TYPE Recipe :
STRUCT
	aRecipe		: ARRAY[1..GVL_CONSTANT.MaxRecipeStep] OF RecipeStep; //Recipe Structure
	iRcpTotalStep			: INT; //Recip Total Number
	control : RecipeControl;
END_STRUCT
END_TYPE

(* stored: Version 1.1.0.1, ProductVersion 3.1.4026.11
   DUT Recipe: Id {a4f709e4-1959-4928-bf7a-7de8f71e6e3e} *)
